PROGRAM MAIN_TECHNOLOGY
VAR
    _technology : Technology;
END_VAR

_technology.Run();

END_PROGRAM

(* stored: Version 1.1.0.1, ProductVersion 3.1.4024.9
   POU MAIN_TECHNOLOGY: Id {c2bf5f61-d736-08ce-0dfa-fcb1ab9b7594}, SpecialFunc None *)
